(* PLC project SafeLOGIC-1, BrAutomation SafeDESIGNER  4.3.4.4 *)
(* stored: companyURL http://www.br-automation.com, creationDateTime Tue Dec 17 14:03:29 2019 *)

PROGRAM Main
  VAR  (* added by the conversion: wires and edge detectors of the diagram *)
    _SAFEBOOL_TO_BOOL77_OUT : BOOL;
  END_VAR

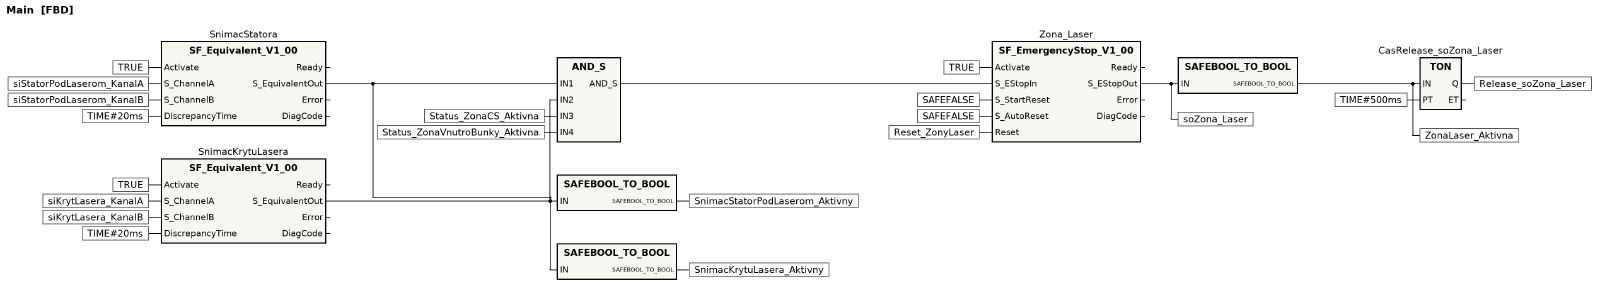
(* FBD diagram, written out as Structured Text *)
SnimacStatora(Activate := TRUE, S_ChannelA := siStatorPodLaserom_KanalA, S_ChannelB := siStatorPodLaserom_KanalB, DiscrepancyTime := TIME#20ms);
SnimacKrytuLasera(Activate := TRUE, S_ChannelA := siKrytLasera_KanalA, S_ChannelB := siKrytLasera_KanalB, DiscrepancyTime := TIME#20ms);
Zona_Laser(Activate := TRUE, S_EStopIn := AND_S(SnimacStatora.S_EquivalentOut, SnimacKrytuLasera.S_EquivalentOut, Status_ZonaCS_Aktivna, Status_ZonaVnutroBunky_Aktivna), S_StartReset := SAFEFALSE, S_AutoReset := SAFEFALSE, Reset := Reset_ZonyLaser);
soZona_Laser := Zona_Laser.S_EStopOut;
SnimacStatorPodLaserom_Aktivny := SAFEBOOL_TO_BOOL(SnimacStatora.S_EquivalentOut);
_SAFEBOOL_TO_BOOL77_OUT := SAFEBOOL_TO_BOOL(Zona_Laser.S_EStopOut);
CasRelease_soZona_Laser(IN := _SAFEBOOL_TO_BOOL77_OUT, PT := TIME#500ms);
Release_soZona_Laser := CasRelease_soZona_Laser.Q;
ZonaLaser_Aktivna := _SAFEBOOL_TO_BOOL77_OUT;
SnimacKrytuLasera_Aktivny := SAFEBOOL_TO_BOOL(SnimacKrytuLasera.S_EquivalentOut);
END_PROGRAM
